// TIA Portal V20 export
// export: Created 2025-12-01T14:57:11.0203502Z, ExportSetting None, DisplayName Totally Integrated Automation Portal, DisplayVersion V20 Update 3, DisplayName TIA Portal Openness, DisplayVersion V20 Update 3, DisplayName TIA Portal Version Control Interface, DisplayVersion V20 Update 3, DisplayName STEP 7 Professional, DisplayVersion V20 Update 3, DisplayName STEP 7 Safety, DisplayVersion V20 Update 2, DisplayName WinCC Basic/Comfort/Advanced, DisplayVersion V20 Update 3, DisplayName WinCC Professional, DisplayVersion V20 Update 3, DisplayName WinCC Unified, DisplayVersion V20 Update 3
FUNCTION "FC724_CambiarUT_DeMesa" : Void   // FC724, LAD
TITLE = "CambiarUT_DeMesa"
{ S7_Optimized_Access := 'FALSE' }
AUTHOR : TRACKING
NAME : 20130301
VERSION : 3.0
// stored: AutoNumber false, SetENOAutomatically false
   VAR_INPUT
      NumeroUT : UInt;   // Numero de UT
      NuevaMesa : UInt;   // Nueva Mesa (En PLC) a insertar UT (Al final de la Cola)
      AlPrincipio : Bool;   // Insertar Al principio de la Nueva Mesa
   END_VAR
   VAR_TEMP
      UT_Anterior : UInt;
      UT_Siguiente : UInt;
      Mesa : UInt;
   END_VAR
BEGIN

NETWORK
TITLE = Inicilizar
////////////////////////////////////////////////////////////////////////
////////////////////////////////////////////////////////////////////////
////////////////////////////////////////////////////////////////////////
// Inicilizar





NETWORK
TITLE = Sacar la UT de la Mesa Antigua
////////////////////////////////////////////////////////////////////////
////////////////////////////////////////////////////////////////////////
////////////////////////////////////////////////////////////////////////
// Sacar de la Mesa Antigua
      L     "DB812_UTs_Control".UT[#NumeroUT].MesaActual;
      L     "CTE_OffsetMesa";
      -I;
      T     #Mesa;

      L     "DB812_UTs_Control".UT[#NumeroUT].UT_AnteriorMesa;
      T     #UT_Anterior;
      L     "DB812_UTs_Control".UT[#NumeroUT].UT_SiguienteMesa;
      T     #UT_Siguiente;

      L     0;  // Inicializo
      T     "DB812_UTs_Control".UT[#NumeroUT].UT_AnteriorMesa;
      T     "DB812_UTs_Control".UT[#NumeroUT].UT_SiguienteMesa;




NETWORK
TITLE = --- Modificar Datos de la UT Anterior
////////////////////////////////////////////////////////////////////////
////////////////////////////////////////////////////////////////////////
////////////////////////////////////////////////////////////////////////
// Modificar Datos de la UT Anterior

      L     #UT_Anterior;
      L     0;  // Primera de la mesa
      <>I;
      JC    NoPrimeraUT_AnteriorUT_EnColaMesaOrigen;
      JU    PrimeraUT_AnteriorUT_EnColaMesaOrigen;


////////////////////////////////////////////////////////////////////////
// No existe ninguna UT Anterior en la Mesa Origen : Era la Primera
PrimeraUT_AnteriorUT_EnColaMesaOrigen:NOP   0;
      L     #UT_Siguiente;
      T     "DB810_ColasMesas".Colas[#Mesa].UT_PrimeraMesa;

      JU    Final_AnteriorUT_EnColaMesaOrigen;


////////////////////////////////////////////////////////////////////////
// Si existe UT Anterior en la Mesa Origen: No Era la Primera
NoPrimeraUT_AnteriorUT_EnColaMesaOrigen:NOP   0;
      L     #UT_Siguiente;
      T     "DB812_UTs_Control".UT[#UT_Anterior].UT_SiguienteMesa;

      JU    Final_AnteriorUT_EnColaMesaOrigen;


////////////////////////////////////////////////////////////////////////
// Final de la Modificacion de la Anterior UT
Final_AnteriorUT_EnColaMesaOrigen:NOP   0;



NETWORK
TITLE = --- Modificar Datos de la UT Siguiente
////////////////////////////////////////////////////////////////////////
////////////////////////////////////////////////////////////////////////
////////////////////////////////////////////////////////////////////////
// Modificar Datos de la UT Siguiente

      L     #UT_Siguiente;
      L     0;  // Es la ultima de la mesa
      ==I;
      JC    UltimaUT_SiguienteUT_EnColaMesaOrigen;
      JU    NoUltimaUT_SiguienteUT_EnColaMesaOrigen;


////////////////////////////////////////////////////////////////////////
// Si existe UT Siguiente en la Mesa Origen: No es la Ultima
UltimaUT_SiguienteUT_EnColaMesaOrigen:NOP   0;
      JU    Final_SiguienteUT_EnColaMesaOrigen;


////////////////////////////////////////////////////////////////////////
// Si existe UT Siguiente en la Mesa Origen: No es la Ultima
NoUltimaUT_SiguienteUT_EnColaMesaOrigen:NOP   0;
      L     #UT_Anterior;
      T     "DB812_UTs_Control".UT[#UT_Siguiente].UT_AnteriorMesa;

      JU    Final_SiguienteUT_EnColaMesaOrigen;


////////////////////////////////////////////////////////////////////////
// Final de la Modificacion de la Anterior UT
Final_SiguienteUT_EnColaMesaOrigen:NOP   0;




NETWORK
TITLE = Poner la UT en la Mesa Nueva
////////////////////////////////////////////////////////////////////////
////////////////////////////////////////////////////////////////////////
////////////////////////////////////////////////////////////////////////

      L     #NuevaMesa;
      T     #Mesa;


////////////////////////////////////////////////////////////////////////
////////////////////////////////////////////////////////////////////////
// --- Donde Hay que insertarlo al Principio o al Final de la Mesa

      SET;
      A     #AlPrincipio;  // Esta Activado ?
      JC    Insertar_PRINCIPIO_EnColaMesaDestino;  // Insertar al Principio de la Mesa
      JU    Insertar_FINAL_EnColaMesaDestino;  // Insertar al Final de la Mesa



NETWORK
TITLE = --- Insertar la UT al FINAL de la Mesa Nueva
////////////////////////////////////////////////////////////////////////
////////////////////////////////////////////////////////////////////////
////////////////////////////////////////////////////////////////////////
// Insertar la UT al FINAL de la Mesa Nueva
Insertar_FINAL_EnColaMesaDestino:NOP   0;
      L     "DB810_ColasMesas".Colas[#Mesa].UT_PrimeraMesa;
      L     0;  // Hay alguna UT en la Mesa
      <>I;
      JC    ExisteUT_FINAL_EnColaMesaDEstino;
      JU    NoExisteUT_FINAL_EnColaMesaDEstino;


////////////////////////////////////////////////////////////////////////
////////////////////////////////////////////////////////////////////////
// No Hay UTs en la Mesa --> Sera la primera UT de la Mesa
NoExisteUT_FINAL_EnColaMesaDEstino:NOP   0;
      L     #NumeroUT;  // Es la primera de la Mesa
      T     "DB810_ColasMesas".Colas[#Mesa].UT_PrimeraMesa;

      L     0;  // Es Unica UT en la Mesa
      T     "DB812_UTs_Control".UT[#NumeroUT].UT_AnteriorMesa;
      T     "DB812_UTs_Control".UT[#NumeroUT].UT_SiguienteMesa;

      L     #NuevaMesa;
      L     "CTE_OffsetMesa";  // Mesa para la Base de Datos
      +I;  // + Offset
      T     "DB812_UTs_Control".UT[#NumeroUT].MesaActual;

      JU    Final_Funcion;


////////////////////////////////////////////////////////////////////////
////////////////////////////////////////////////////////////////////////
// Hay UTs en la Mesa --> Sera la ultima UT de la Mesa
ExisteUT_FINAL_EnColaMesaDEstino:NOP   0;
      L     "DB810_ColasMesas".Colas[#Mesa].UT_PrimeraMesa;
      T     #UT_Siguiente;


////////////////////////////////////////////////////////////////////////
// Buscar ultima UT de la Mesa
BucleBusquedaUltimaUT_FINAL_EnColaMesaDestino:NOP   0;
      L     "DB812_UTs_Control".UT[#UT_Siguiente].UT_SiguienteMesa;
      L     0;  // Ultima UT
      ==I;
      JC    EncontradaUltimaUT_FINAL_EncolaMesaDestino;

      L     "DB812_UTs_Control".UT[#UT_Siguiente].UT_SiguienteMesa;
      T     #UT_Siguiente;

      JU    BucleBusquedaUltimaUT_FINAL_EnColaMesaDestino;


////////////////////////////////////////////////////////////////////////
// Ya esta encontrada la ultima UT en la Mesa
// Primero se modifica la Ultima UT de la mesa
// Segundo se modifica la UT a insertar
EncontradaUltimaUT_FINAL_EncolaMesaDestino:NOP   0;

// Modificar la Ultima UT de la Mesa
      L     #NumeroUT;
      T     "DB812_UTs_Control".UT[#UT_Siguiente].UT_SiguienteMesa;


// Modificar la UT a Insertar
      L     #UT_Siguiente;
      T     "DB812_UTs_Control".UT[#NumeroUT].UT_AnteriorMesa;
      L     0;
      T     "DB812_UTs_Control".UT[#NumeroUT].UT_SiguienteMesa;

      L     #NuevaMesa;
      L     "CTE_OffsetMesa";  // Mesa para la Base de Datos
      +I;  // + Offset
      T     "DB812_UTs_Control".UT[#NumeroUT].MesaActual;

      JU    Final_Funcion;



NETWORK
TITLE = --- Insertar la UT al PRINCIPIO de la Mesa Nueva
// Buscar el final de la Mesa 
// Modificar datos de la cola
////////////////////////////////////////////////////////////////////////
////////////////////////////////////////////////////////////////////////
////////////////////////////////////////////////////////////////////////
// Insertar la UT al PRINCIPIO de la Mesa Nueva
Insertar_PRINCIPIO_EnColaMesaDestino:NOP   0;
      L     "DB810_ColasMesas".Colas[#Mesa].UT_PrimeraMesa;
      T     #UT_Siguiente;

      L     #UT_Siguiente;
      L     0;  // Hay alguna UT en la Mesa
      <>I;
      JC    ExisteUT_PRINCIPIO_EnColaMesaDestino;
      JU    NoExisteUT_PRINCIPIO_EnColaMesaDestino;



////////////////////////////////////////////////////////////////////////
////////////////////////////////////////////////////////////////////////
// --- NO Hay alguna UT en la Mesa
// --- Hay que ponerla al principio de la Mesa
NoExisteUT_PRINCIPIO_EnColaMesaDestino:NOP   0;
      L     #NumeroUT;  // Es la primera de la Mesa
      T     "DB810_ColasMesas".Colas[#Mesa].UT_PrimeraMesa;

      L     0;  // Es Unica UT en la Mesa
      T     "DB812_UTs_Control".UT[#NumeroUT].UT_AnteriorMesa;
      T     "DB812_UTs_Control".UT[#NumeroUT].UT_SiguienteMesa;

      L     #NuevaMesa;
      L     "CTE_OffsetMesa";  // Mesa para la Base de Datos
      +I;  // + Offset
      T     "DB812_UTs_Control".UT[#NumeroUT].MesaActual;

      JU    Final_Funcion;


////////////////////////////////////////////////////////////////////////
////////////////////////////////////////////////////////////////////////
// --- Hay alguna UT en la Mesa
// --- Hay que ponerla al principio de la Mesa
ExisteUT_PRINCIPIO_EnColaMesaDestino:NOP   0;
      L     #NumeroUT;  // Es la primera de la Mesa
      T     "DB810_ColasMesas".Colas[#Mesa].UT_PrimeraMesa;

      L     0;  // Es Unica UT en la Mesa
      T     "DB812_UTs_Control".UT[#NumeroUT].UT_AnteriorMesa;
      L     #UT_Siguiente;  // El que estaba primero
      T     "DB812_UTs_Control".UT[#NumeroUT].UT_SiguienteMesa;

      L     #NuevaMesa;
      L     "CTE_OffsetMesa";  // Mesa para la Base de Datos
      +I;  // + Offset
      T     "DB812_UTs_Control".UT[#NumeroUT].MesaActual;


////////////////////////////////////////////////////////////////////////
// Modificar que estaba primero
      L     #NumeroUT;  // Aviso del que estaba primero
      T     "DB812_UTs_Control".UT[#UT_Siguiente].UT_AnteriorMesa;


      JU    Final_Funcion;



NETWORK
TITLE = Final de la funcion
Final_Funcion:NOP   0;


END_FUNCTION
